KUKA KRL program: masref_user.src, masref_user.dat

--- masref_user.src ---
&ACCESS RV
&REL 1
&COMMENT Mastering Reference User Program
&PARAM DISKPATH = KRC:\R1\Program
DEF MasRef_USER()
END

GLOBAL DEF MASREFSTARTG1()
;FOLD Teach path and position for reference group 1
;ENDFOLD

END

GLOBAL DEF MASREFBACKG1()
;FOLD Teach path back for reference group 1
;ENDFOLD

END

GLOBAL DEF MASREFSTARTG2()
;FOLD Teach path and position for reference group 2
;ENDFOLD

END

GLOBAL DEF MASREFBACKG2()
;FOLD Teach path back for reference group 2
;ENDFOLD

END

GLOBAL DEF MASREFSTARTG3()
;FOLD Teach path and position for reference group 3
;ENDFOLD

END

GLOBAL DEF MASREFBACKG3()
;FOLD Teach path back for reference group 3
;ENDFOLD

END

--- masref_user.dat ---
&ACCESS RV
&COMMENT Mastering Reference User Program
&PARAM DISKPATH = KRC:\R1\Program
&PARAM TEMPLATE = C:\KRC\Roboter\Template\vorgabe
&PARAM EDITMASK = *
DEFDAT MasRef_User PUBLIC
;FOLD EXTERNAL DECLARATIONS;%{PE}%MKUKATPBASIS,%CEXT,%VCOMMON,%P
;FOLD BASISTECH EXT;%{PE}%MKUKATPBASIS,%CEXT,%VEXT,%P
  EXT  BAS (BAS_COMMAND  :IN,REAL  :IN )
;ENDFOLD (BASISTECH EXT)
;FOLD USER EXT;%{E}%MKUKATPUSER,%CEXT,%VEXT,%P
;Make here your modifications

;ENDFOLD (USER EXT)
;ENDFOLD (EXTERNAL DECLERATIONS)
;FOLD reference groups
; order of master reference group number in array is of no relevance, but group "1" is required
; "0" means no master reference test
; "1" means group number for robot axes and robroot kinematic axes
; "2", "3" means group number of external kinematic axes
DECL GLOBAL CONST INT MASREFg_GroupSequence[3] ; contains reference groups to test
MASREFg_GroupSequence[1]=1
MASREFg_GroupSequence[2]=0
MASREFg_GroupSequence[3]=0
;ENDFOLD (reference groups)
ENDDAT
